PROGRAM uloha2
VAR
	M1: BOOL;
	M2: BOOL;
	M3: BOOL;
	start1: BOOL;
	start2: BOOL;
	start3: BOOL;
	stav: INT;
	pocet_motorov: INT;
	stop: BOOL;
END_VAR


pocet_motorov := 0;

IF M1 = TRUE THEN
    pocet_motorov := pocet_motorov + 1;
END_IF;

IF M2 = TRUE THEN
    pocet_motorov := pocet_motorov + 1;
END_IF;

IF M3 = TRUE THEN
    pocet_motorov := pocet_motorov + 1;
END_IF;



CASE stav OF

    0:  
        IF start1 = TRUE THEN
            M1 := TRUE;
            stav := 1;
        ELSIF start2 = TRUE THEN
            M2 := TRUE;
            stav := 1;
        ELSIF start3 = TRUE THEN
            M3 := TRUE;
            stav := 1;
        END_IF;


    1:  
        IF pocet_motorov >= 2 THEN
            stav := 2;
        ELSE
            IF start1 = TRUE AND NOT M1 = TRUE THEN
                M1 := TRUE;
            END_IF;

            IF start2 = TRUE AND NOT M2 = TRUE  THEN
                M2 := TRUE;
            END_IF;

            IF start3 = TRUE AND NOT M3 = TRUE THEN
                M3 := TRUE;
            END_IF;
        END_IF;


    2:  
        IF pocet_motorov < 2 THEN
            stav := 1;
        END_IF;

END_CASE;



IF stop THEN
    M1 := FALSE;
    M2 := FALSE;
    M3 := FALSE;
    pocet_motorov := 0;
    stav := 0;
	start1 := FALSE;
	start2 := FALSE;
	start3 := FALSE;
	stop := FALSE;
END_IF;

END_PROGRAM

(* stored: Version 1.1.0.1
   POU uloha2: Id {fab15751-bfe8-4461-ab23-500ac923cd79}, SpecialFunc None *)
